// Mitsubishi GX Works2 project: 20   PLC: FX3G

// task Task_01 (event TRUE, interval 0, priority 31): POU_01

PROGRAM POU_01
VAR
  wstep : INT;
  ton1 : TON;
END_VAR
M99 := FALSE AND
M0 AND M1 AND M2 AND
Y1 AND Y2 AND Y3 AND Y4;

IF M8002 THEN
	wstep := 0;
END_IF;

CASE wstep OF
	0:
		ZRST(TRUE, Y1, Y4);
		
		IF M0 THEN
			wstep := 20;
		END_IF;
		
	20:
		Y3 := TRUE;
		Y4 := TRUE;
		
		IF M2 THEN
			wstep := 21;
		END_IF;
		IF M1 THEN
			wstep := 22;
		END_IF;
	21:
		Y2 := TRUE;
		Y3 := FALSE;
		ton1(in := NOT ton1.q, pt := t#5s);
		
		IF ton1.q THEN
			wstep := 0;
		END_IF;		
	22:
		Y1 := TRUE;
		Y4 := FALSE;
		ton1(in := NOT ton1.q, pt := t#5s);

		IF ton1.q THEN
			wstep := 0;
		END_IF;
END_CASE;
END_PROGRAM
